FUNCTION Convert_REAL_TO_TOD : Hresult
VAR_INPUT
	in : REAL;
	out : REFERENCE TO TOD;
END_VAR
VAR
	converted : TOD;
END_VAR
VAR CONSTANT
	INCOMPATIBLE : HRESULT := 16#9811070E;
END_VAR

converted := REAL_TO_TOD(in);

IF (TOD_TO_REAL(converted) <> in) THEN
	Convert_REAL_TO_TOD := INCOMPATIBLE;
	RETURN;
END_IF

out := converted;

END_FUNCTION

(* stored: Version 1.1.0.1, ProductVersion 3.1.4024.12
   POU Convert_REAL_TO_TOD: Id {1705d395-b890-4432-897c-0bf50aea5f47}, SpecialFunc None *)
